{attribute 'GeneratedUsingTerminal: EM7004-0000-0017'}
{attribute addProperty BoxType "EM7004-0000-0017"}
{attribute addProperty Id "StatusAT %I*Status_882A150F2"}
{attribute addProperty CRC "1707713494"}
{attribute addProperty Size "2"}
TYPE PLS_Inputs_65C9A3D6 EXTENDS InputBase_8311D824 :
STRUCT
	{attribute addProperty Name "Status"}
	Status AT %I* : Status_882A150F;
END_STRUCT
END_TYPE
